				Clear(STRUCT_ALIGNMENT2);
				STRUCT_ALIGNMENT2.aBool := TRUE; STRUCT_ALIGNMENT2.aInt := -1; STRUCT_ALIGNMENT2.aUint := 2;
				STRUCT_ALIGNMENT2.Bools[0] := TRUE; STRUCT_ALIGNMENT2.Bools[3] := TRUE;
				iVarBinSize := ToAryByte(In:=STRUCT_ALIGNMENT2, Order:=_eBYTE_ORDER#_LOW_HIGH, AryOut:=iVarBin[0]);
				Inc(iVarIndex);
			211:
				iVarName := 'STRUCT_ALIGNMENT2_ARR_D1';
				iVarDeclare := 'ARRAY[0..2] OF Alignment2Struct';
				iVarValue := '[{"aBool":true, "aInt":-1, "aUint":2, "Bools":[true,false,false,true]}, {"aBool":false, "aInt":0, "aUint":0, "Bools":[false,false,false,false]}, {"aBool":true, "aInt":-1, "aUint":2, "Bools":[true,false,false,true]}]';
				iVarKsType := 'alignment2_struct_t::alignment2_struct_array_1d(3)';
				iVarKsId := 'struct_alignment2_arr_d1';
				
				Clear(STRUCT_ALIGNMENT2);
				STRUCT_ALIGNMENT2.aBool := TRUE; STRUCT_ALIGNMENT2.aInt := -1; STRUCT_ALIGNMENT2.aUint := 2;
				STRUCT_ALIGNMENT2.Bools[0] := TRUE; STRUCT_ALIGNMENT2.Bools[3] := TRUE;
				Clear(STRUCT_ALIGNMENT2_ARR_D1);
				STRUCT_ALIGNMENT2_ARR_D1[0] := STRUCT_ALIGNMENT2; STRUCT_ALIGNMENT2_ARR_D1[2] := STRUCT_ALIGNMENT2;
				
				iVarBinSize := ToAryByte(In:=STRUCT_ALIGNMENT2_ARR_D1, Order:=_eBYTE_ORDER#_LOW_HIGH, AryOut:=iVarBin[0]);
				iVarIndex := iVarIndex - iVarIndex MOD 10 + 10;

			// Alignment4Struct
			220:
				iVarName := 'STRUCT_ALIGNMENT4';
				iVarDeclare := 'Alignment4Struct';
				iVarValue := '{"aUdint":1, "aDint":-2, "Uints":[3,4], "Bytes":[5,6,7,8]}';
				iVarKsType := 'alignment4_struct_t::alignment4_struct';
				iVarKsId := 'struct_alignment4';
				
				Clear(STRUCT_ALIGNMENT4);
				STRUCT_ALIGNMENT4.aUdint := 1; STRUCT_ALIGNMENT4.aDint := -2;
				STRUCT_ALIGNMENT4.Uints[0] := 3; STRUCT_ALIGNMENT4.Uints[1] := 4;
				STRUCT_ALIGNMENT4.Bytes[0] := 5; STRUCT_ALIGNMENT4.Bytes[1] := 6; STRUCT_ALIGNMENT4.Bytes[2] := 7; STRUCT_ALIGNMENT4.Bytes[3] := 8;
				iVarBinSize := ToAryByte(In:=STRUCT_ALIGNMENT4, Order:=_eBYTE_ORDER#_LOW_HIGH, AryOut:=iVarBin[0]);
				iVarIndex := iVarIndex - iVarIndex MOD 10 + 10;
				
			// Alignment8Struct
			230:
				iVarName := 'STRUCT_ALIGNMENT8';
				iVarDeclare := 'Alignment8Struct';
				iVarValue := '{"aUlint":1, "aLint":-2, "Udints":[3,4], "aAlignment2Struct":{"aBool":true, "aInt":-1, "aUint":2, "Bools":[true,false,false,true]}}';
				iVarKsType := 'alignment8_struct_t::alignment8_struct';
				iVarKsId := 'struct_alignment8';
				
				Clear(STRUCT_ALIGNMENT8);
				STRUCT_ALIGNMENT8.aUlint := 1; STRUCT_ALIGNMENT8.aLint := -2;
				STRUCT_ALIGNMENT8.Udints[0] := 3; STRUCT_ALIGNMENT8.Udints[1] := 4;
				Clear(STRUCT_ALIGNMENT2);
				STRUCT_ALIGNMENT2.aBool := TRUE; STRUCT_ALIGNMENT2.aInt := -1; STRUCT_ALIGNMENT2.aUint := 2;
				STRUCT_ALIGNMENT2.Bools[0] := TRUE; STRUCT_ALIGNMENT2.Bools[3] := TRUE;
				STRUCT_ALIGNMENT8.aAlignment2Struct := STRUCT_ALIGNMENT2;
				iVarBinSize := ToAryByte(In:=STRUCT_ALIGNMENT8, Order:=_eBYTE_ORDER#_LOW_HIGH, AryOut:=iVarBin[0]);
				iVarIndex := iVarIndex - iVarIndex MOD 10 + 10;
			
			// SmallStruct
			240:
				iVarName := 'STRUCT_SMALL_LH';
				iVarDeclare := 'SmallStruct';
				iVarValue := '{"s":"a","u":1}';
				iVarKsType := 'small_struct_t::small_struct';
				iVarKsId := 'struct_small_lh';
				
				Clear(STRUCT_SMALL);
				STRUCT_SMALL.u := 1; STRUCT_SMALL.s := 'a';
				iVarBinSize := ToAryByte(In:=STRUCT_SMALL, Order:=_eBYTE_ORDER#_LOW_HIGH, AryOut:=iVarBin[0]);
				Inc(iVarIndex);
			241:
				iVarName := 'STRUCT_SMALL_ARR_D1_LH';
				iVarDeclare := 'ARRAY[0..2] OF SmallStruct';
				iVarValue := '[{"s":"a","u":1},{"s":"b","u":2},{"s":"c","u":3}]';
				iVarKsType := 'small_struct_t::small_struct_array_1d(3)';
				iVarKsId := 'struct_small_arr_d1_lh';
				
				Clear(STRUCT_SMALL_ARR_D1);
				STRUCT_SMALL_ARR_D1[0].u := 1; STRUCT_SMALL_ARR_D1[0].s := 'a';
				STRUCT_SMALL_ARR_D1[1].u := 2; STRUCT_SMALL_ARR_D1[1].s := 'b';
				STRUCT_SMALL_ARR_D1[2].u := 3; STRUCT_SMALL_ARR_D1[2].s := 'c';
				iVarBinSize := ToAryByte(In:=STRUCT_SMALL_ARR_D1, Order:=_eBYTE_ORDER#_LOW_HIGH, AryOut:=iVarBin[0]);
				Inc(iVarIndex);
			242:
				iVarName := 'STRUCT_SMALL_ARR_D2_LH';
				iVarDeclare := 'ARRAY[0..2,0..2] OF SmallStruct';
				iVarValue := '[[{"s":"a","u":1},{"s":"b","u":2},{"s":"c","u":3}],[{"s":"d","u":4},{"s":"e","u":5},{"s":"f","u":6}],[{"s":"g","u":7},{"s":"h","u":8},{"s":"i","u":9}]]';
				iVarKsType := 'small_struct_t::small_struct_array_2d(3,3)';
				iVarKsId := 'struct_small_arr_d2_lh';
				
				Clear(STRUCT_SMALL_ARR_D2);
				STRUCT_SMALL_ARR_D2[0, 0].u := 1; STRUCT_SMALL_ARR_D2[0, 0].s := 'a';
				STRUCT_SMALL_ARR_D2[0, 1].u := 2; STRUCT_SMALL_ARR_D2[0, 1].s := 'b';
				STRUCT_SMALL_ARR_D2[0, 2].u := 3; STRUCT_SMALL_ARR_D2[0, 2].s := 'c';
				STRUCT_SMALL_ARR_D2[1, 0].u := 4; STRUCT_SMALL_ARR_D2[1, 0].s := 'd';
				STRUCT_SMALL_ARR_D2[1, 1].u := 5; STRUCT_SMALL_ARR_D2[1, 1].s := 'e';
				STRUCT_SMALL_ARR_D2[1, 2].u := 6; STRUCT_SMALL_ARR_D2[1, 2].s := 'f';
				STRUCT_SMALL_ARR_D2[2, 0].u := 7; STRUCT_SMALL_ARR_D2[2, 0].s := 'g';
				STRUCT_SMALL_ARR_D2[2, 1].u := 8; STRUCT_SMALL_ARR_D2[2, 1].s := 'h';
				STRUCT_SMALL_ARR_D2[2, 2].u := 9; STRUCT_SMALL_ARR_D2[2, 2].s := 'i';
				iVarBinSize := ToAryByte(In:=STRUCT_SMALL_ARR_D2, Order:=_eBYTE_ORDER#_LOW_HIGH, AryOut:=iVarBin[0]);
				Inc(iVarIndex);
			243:
				iVarName := 'STRUCT_SMALL_ARR_D3_LH';
				iVarDeclare := 'ARRAY[0..2,0..2,0..2] OF SmallStruct';
				iVarValue := '[[[{"s":"a","u":1},{"s":"b","u":2},{"s":"c","u":3}],[{"s":"d","u":4},{"s":"e","u":5},{"s":"f","u":6}],[{"s":"g","u":7},{"s":"h","u":8},{"s":"i","u":9}]],[[{"s":"j","u":10},{"s":"k","u":11},{"s":"l","u":12}],[{"s":"m","u":13},{"s":"n","u":14},{"s":"o","u":15}],[{"s":"p","u":16},{"s":"q","u":17},{"s":"r","u":18}]],[[{"s":"s","u":19},{"s":"t","u":20},{"s":"u","u":21}],[{"s":"v","u":22},{"s":"w","u":23},{"s":"x","u":24}],[{"s":"y","u":25},{"s":"z","u":26},{"s":"0","u":27}]]]';
				iVarKsType := 'small_struct_t::small_struct_array_3d(3,3,3)';
				iVarKsId := 'struct_small_arr_d3_lh';
				
				Clear(STRUCT_SMALL_ARR_D3);
				STRUCT_SMALL_ARR_D3[0, 0, 0].u := 1; STRUCT_SMALL_ARR_D3[0, 0, 0].s := 'a';
				STRUCT_SMALL_ARR_D3[0, 0, 1].u := 2; STRUCT_SMALL_ARR_D3[0, 0, 1].s := 'b';
				STRUCT_SMALL_ARR_D3[0, 0, 2].u := 3; STRUCT_SMALL_ARR_D3[0, 0, 2].s := 'c';
				STRUCT_SMALL_ARR_D3[0, 1, 0].u := 4; STRUCT_SMALL_ARR_D3[0, 1, 0].s := 'd';
				STRUCT_SMALL_ARR_D3[0, 1, 1].u := 5; STRUCT_SMALL_ARR_D3[0, 1, 1].s := 'e';
				STRUCT_SMALL_ARR_D3[0, 1, 2].u := 6; STRUCT_SMALL_ARR_D3[0, 1, 2].s := 'f';
				STRUCT_SMALL_ARR_D3[0, 2, 0].u := 7; STRUCT_SMALL_ARR_D3[0, 2, 0].s := 'g';
				STRUCT_SMALL_ARR_D3[0, 2, 1].u := 8; STRUCT_SMALL_ARR_D3[0, 2, 1].s := 'h';
				STRUCT_SMALL_ARR_D3[0, 2, 2].u := 9; STRUCT_SMALL_ARR_D3[0, 2, 2].s := 'i';
				STRUCT_SMALL_ARR_D3[1, 0, 0].u := 10; STRUCT_SMALL_ARR_D3[1, 0, 0].s := 'j';
				STRUCT_SMALL_ARR_D3[1, 0, 1].u := 11; STRUCT_SMALL_ARR_D3[1, 0, 1].s := 'k';
				STRUCT_SMALL_ARR_D3[1, 0, 2].u := 12; STRUCT_SMALL_ARR_D3[1, 0, 2].s := 'l';
				STRUCT_SMALL_ARR_D3[1, 1, 0].u := 13; STRUCT_SMALL_ARR_D3[1, 1, 0].s := 'm';
				STRUCT_SMALL_ARR_D3[1, 1, 1].u := 14; STRUCT_SMALL_ARR_D3[1, 1, 1].s := 'n';
				STRUCT_SMALL_ARR_D3[1, 1, 2].u := 15; STRUCT_SMALL_ARR_D3[1, 1, 2].s := 'o';
				STRUCT_SMALL_ARR_D3[1, 2, 0].u := 16; STRUCT_SMALL_ARR_D3[1, 2, 0].s := 'p';
				STRUCT_SMALL_ARR_D3[1, 2, 1].u := 17; STRUCT_SMALL_ARR_D3[1, 2, 1].s := 'q';
				STRUCT_SMALL_ARR_D3[1, 2, 2].u := 18; STRUCT_SMALL_ARR_D3[1, 2, 2].s := 'r';
				STRUCT_SMALL_ARR_D3[2, 0, 0].u := 19; STRUCT_SMALL_ARR_D3[2, 0, 0].s := 's';
				STRUCT_SMALL_ARR_D3[2, 0, 1].u := 20; STRUCT_SMALL_ARR_D3[2, 0, 1].s := 't';
				STRUCT_SMALL_ARR_D3[2, 0, 2].u := 21; STRUCT_SMALL_ARR_D3[2, 0, 2].s := 'u';
				STRUCT_SMALL_ARR_D3[2, 1, 0].u := 22; STRUCT_SMALL_ARR_D3[2, 1, 0].s := 'v';
				STRUCT_SMALL_ARR_D3[2, 1, 1].u := 23; STRUCT_SMALL_ARR_D3[2, 1, 1].s := 'w';
				STRUCT_SMALL_ARR_D3[2, 1, 2].u := 24; STRUCT_SMALL_ARR_D3[2, 1, 2].s := 'x';
				STRUCT_SMALL_ARR_D3[2, 2, 0].u := 25; STRUCT_SMALL_ARR_D3[2, 2, 0].s := 'y';
				STRUCT_SMALL_ARR_D3[2, 2, 1].u := 26; STRUCT_SMALL_ARR_D3[2, 2, 1].s := 'z';
				STRUCT_SMALL_ARR_D3[2, 2, 2].u := 27; STRUCT_SMALL_ARR_D3[2, 2, 2].s := '0';
				iVarBinSize := ToAryByte(In:=STRUCT_SMALL_ARR_D3, Order:=_eBYTE_ORDER#_LOW_HIGH, AryOut:=iVarBin[0]);
				Inc(iVarIndex);
			244:
				iVarName := 'STRUCT_SMALL_ARR_D1_E1_LH';
				iVarDeclare := 'ARRAY[0..0] OF SmallStruct';
				iVarValue := '[{"s":"a","u":1}]';
				iVarKsType := 'small_struct_t::small_struct_array_1d(1)';
				iVarKsId := 'struct_small_arr_d1_e1_lh';
				
				Clear(STRUCT_SMALL_ARR_D1_E1);
				STRUCT_SMALL_ARR_D1_E1[0].u := 1; STRUCT_SMALL_ARR_D1_E1[0].s := 'a';
				iVarBinSize := ToAryByte(In:=STRUCT_SMALL_ARR_D1_E1, Order:=_eBYTE_ORDER#_LOW_HIGH, AryOut:=iVarBin[0]);
				Inc(iVarIndex);
			245:
				iVarName := 'STRUCT_SMALL_ARR_D2_E1_LH';
				iVarDeclare := 'ARRAY[0..0,0..0] OF SmallStruct';
				iVarValue := '[[{"s":"a","u":1}]]';
				iVarKsType := 'small_struct_t::small_struct_array_2d(1,1)';
				iVarKsId := 'struct_small_arr_d2_e1_lh';
				
				Clear(STRUCT_SMALL_ARR_D2_E1);
				STRUCT_SMALL_ARR_D2_E1[0, 0].u := 1; STRUCT_SMALL_ARR_D2_E1[0, 0].s := 'a';
				iVarBinSize := ToAryByte(In:=STRUCT_SMALL_ARR_D2_E1, Order:=_eBYTE_ORDER#_LOW_HIGH, AryOut:=iVarBin[0]);
				Inc(iVarIndex);
			246:
				iVarName := 'STRUCT_SMALL_ARR_D3_E1_LH';
				iVarDeclare := 'ARRAY[0..0,0..0,0..0] OF SmallStruct';
				iVarValue := '[[[{"s":"a","u":1}]]]';
				iVarKsType := 'small_struct_t::small_struct_array_3d(1,1,1)';
				iVarKsId := 'struct_small_arr_d3_e1_lh';
				
				Clear(STRUCT_SMALL_ARR_D3_E1);
				STRUCT_SMALL_ARR_D3_E1[0, 0, 0].u := 1; STRUCT_SMALL_ARR_D3_E1[0, 0, 0].s := 'a';
				iVarBinSize := ToAryByte(In:=STRUCT_SMALL_ARR_D3_E1, Order:=_eBYTE_ORDER#_LOW_HIGH, AryOut:=iVarBin[0]);
				iVarIndex := iVarIndex - iVarIndex MOD 10 + 10;
				
			// PaddedStruct
			250:
				iVarName := 'STRUCT_PADDED_LH';
				iVarDeclare := 'PaddedStruct';
				iVarValue := '{"aUsint":1, "aUint":2, "aSint":-3, "aDint":-4, "aUlint":5, "aBool":true}';
				iVarKsType := 'padded_struct_t::padded_struct';
				iVarKsId := 'struct_padded_lh';
				
				Clear(STRUCT_PADDED);
				STRUCT_PADDED.aUsint := 1; STRUCT_PADDED.aUint := 2; STRUCT_PADDED.aSint := -3;
				STRUCT_PADDED.aDint := -4; STRUCT_PADDED.aUlint := 5; STRUCT_PADDED.aBool := TRUE;
				iVarBinSize := ToAryByte(In:=STRUCT_PADDED, Order:=_eBYTE_ORDER#_LOW_HIGH, AryOut:=iVarBin[0]);
				Inc(iVarIndex);
			251:
				iVarName := 'STRUCT_PADDED_ARR_D1_LH';
				iVarDeclare := 'ARRAY[0..2] OF PaddedStruct';
				iVarValue := '[{"aUsint":1, "aUint":2, "aSint":-3, "aDint":-4, "aUlint":5, "aBool":true}, {"aUsint":6, "aUint":7, "aSint":-8, "aDint":-9, "aUlint":10, "aBool":false}, {"aUsint":11, "aUint":12, "aSint":-13, "aDint":-14, "aUlint":15, "aBool":true}]';
				iVarKsType := 'padded_struct_t::padded_struct_array_1d(3)';
				iVarKsId := 'struct_padded_arr_d1_lh';
				
				Clear(STRUCT_PADDED_ARR_D1);
				STRUCT_PADDED_ARR_D1[0].aUsint := 1; STRUCT_PADDED_ARR_D1[0].aUint := 2; STRUCT_PADDED_ARR_D1[0].aSint := -3;
				STRUCT_PADDED_ARR_D1[0].aDint := -4; STRUCT_PADDED_ARR_D1[0].aUlint := 5; STRUCT_PADDED_ARR_D1[0].aBool := TRUE;
				STRUCT_PADDED_ARR_D1[1].aUsint := 6; STRUCT_PADDED_ARR_D1[1].aUint := 7; STRUCT_PADDED_ARR_D1[1].aSint := -8;
				STRUCT_PADDED_ARR_D1[1].aDint := -9; STRUCT_PADDED_ARR_D1[1].aUlint := 10; STRUCT_PADDED_ARR_D1[1].aBool := FALSE;
				STRUCT_PADDED_ARR_D1[2].aUsint := 11; STRUCT_PADDED_ARR_D1[2].aUint := 12; STRUCT_PADDED_ARR_D1[2].aSint := -13;
				STRUCT_PADDED_ARR_D1[2].aDint := -14; STRUCT_PADDED_ARR_D1[2].aUlint := 15; STRUCT_PADDED_ARR_D1[2].aBool := TRUE;
				iVarBinSize := ToAryByte(In:=STRUCT_PADDED_ARR_D1, Order:=_eBYTE_ORDER#_LOW_HIGH, AryOut:=iVarBin[0]);
				Inc(iVarIndex);
			252:
				iVarName := 'STRUCT_PADDED_ARR_D1_E1_LH';
				iVarDeclare := 'ARRAY[0..0] OF PaddedStruct';
				iVarValue := '[{"aUsint":1, "aUint":2, "aSint":-3, "aDint":-4, "aUlint":5, "aBool":true}]';
				iVarKsType := 'padded_struct_t::padded_struct_array_1d(1)';
				iVarKsId := 'struct_padded_arr_d1_e1_lh';
				
				Clear(STRUCT_PADDED_ARR_D1_E1);
				STRUCT_PADDED_ARR_D1_E1[0].aUsint := 1; STRUCT_PADDED_ARR_D1_E1[0].aUint := 2; STRUCT_PADDED_ARR_D1_E1[0].aSint := -3;
				STRUCT_PADDED_ARR_D1_E1[0].aDint := -4; STRUCT_PADDED_ARR_D1_E1[0].aUlint := 5; STRUCT_PADDED_ARR_D1_E1[0].aBool := TRUE;
				iVarBinSize := ToAryByte(In:=STRUCT_PADDED_ARR_D1_E1, Order:=_eBYTE_ORDER#_LOW_HIGH, AryOut:=iVarBin[0]);
				Inc(iVarIndex);
			253:
				iVarName := 'STRUCT_PADDED_ARR_D2_E1_LH';
				iVarDeclare := 'ARRAY[0..0,0..0] OF PaddedStruct';
				iVarValue := '[[{"aUsint":1, "aUint":2, "aSint":-3, "aDint":-4, "aUlint":5, "aBool":true}]]';
				iVarKsType := 'padded_struct_t::padded_struct_array_2d(1,1)';
				iVarKsId := 'struct_padded_arr_d2_e1_lh';
				
				Clear(STRUCT_PADDED_ARR_D2_E1);
				STRUCT_PADDED_ARR_D2_E1[0, 0].aUsint := 1; STRUCT_PADDED_ARR_D2_E1[0, 0].aUint := 2; STRUCT_PADDED_ARR_D2_E1[0, 0].aSint := -3;
				STRUCT_PADDED_ARR_D2_E1[0, 0].aDint := -4; STRUCT_PADDED_ARR_D2_E1[0, 0].aUlint := 5; STRUCT_PADDED_ARR_D2_E1[0, 0].aBool := TRUE;
				iVarBinSize := ToAryByte(In:=STRUCT_PADDED_ARR_D2_E1, Order:=_eBYTE_ORDER#_LOW_HIGH, AryOut:=iVarBin[0]);
				Inc(iVarIndex);
			254:
				iVarName := 'STRUCT_PADDED_ARR_D3_E1_LH';
				iVarDeclare := 'ARRAY[0..0,0..0,0..0] OF PaddedStruct';
				iVarValue := '[[[{"aUsint":1, "aUint":2, "aSint":-3, "aDint":-4, "aUlint":5, "aBool":true}]]]';
				iVarKsType := 'padded_struct_t::padded_struct_array_3d(1,1,1)';
				iVarKsId := 'struct_padded_arr_d3_e1_lh';
				
				Clear(STRUCT_PADDED_ARR_D3_E1);
				STRUCT_PADDED_ARR_D3_E1[0, 0, 0].aUsint := 1; STRUCT_PADDED_ARR_D3_E1[0, 0, 0].aUint := 2; STRUCT_PADDED_ARR_D3_E1[0, 0, 0].aSint := -3;
				STRUCT_PADDED_ARR_D3_E1[0, 0, 0].aDint := -4; STRUCT_PADDED_ARR_D3_E1[0, 0, 0].aUlint := 5; STRUCT_PADDED_ARR_D3_E1[0, 0, 0].aBool := TRUE;
				iVarBinSize := ToAryByte(In:=STRUCT_PADDED_ARR_D3_E1, Order:=_eBYTE_ORDER#_LOW_HIGH, AryOut:=iVarBin[0]);
				iVarIndex := iVarIndex - iVarIndex MOD 10 + 10;

			// UnionStruct
			260:
				iVarName := 'STRUCT_UNION_LH';
				iVarDeclare := 'UnionStruct';
				// Since Union is not supported, the values ​​of each field are listed separately.
				iVarValue := '{"Alignment1Unions":[{"Bytes":[1,2,3,4]},{"Bytes":[5,6,7,8]}], "Alignment2Unions":[{"aBool":true,"Words":[9,10]}, {"aBool":true,"Words":[11,12]}], "aAlignment4Union":{"Bytes":[13,0,0,0],"Dwords":[13,14]}, "aAlignment8Union":{"Words":[15,0,0,0],"aLword":15}}';
				iVarKsType := 'union_struct_t::union_struct';
				iVarKsId := 'union_struct_lh';
				
				Clear(STRUCT_UNION);
				STRUCT_UNION.Alignment1Unions[0].Bytes[0] := 1; STRUCT_UNION.Alignment1Unions[0].Bytes[1] := 2; STRUCT_UNION.Alignment1Unions[0].Bytes[2] := 3; STRUCT_UNION.Alignment1Unions[0].Bytes[3] := 4;
				STRUCT_UNION.Alignment1Unions[1].Bytes[0] := 5; STRUCT_UNION.Alignment1Unions[1].Bytes[1] := 6; STRUCT_UNION.Alignment1Unions[1].Bytes[2] := 7; STRUCT_UNION.Alignment1Unions[1].Bytes[3] := 8;
				STRUCT_UNION.Alignment2Unions[0].Words[0] := 9; STRUCT_UNION.Alignment2Unions[0].Words[1] := 10;
				STRUCT_UNION.Alignment2Unions[1].Words[0] := 11; STRUCT_UNION.Alignment2Unions[1].Words[1] := 12;
				STRUCT_UNION.aAlignment4Union.Dwords[0] := 13; STRUCT_UNION.aAlignment4Union.Dwords[1] := 14;
				STRUCT_UNION.aAlignment8Union.aLword := 15;
				
				iVarBinSize := ToAryByte(In:=STRUCT_UNION, Order:=_eBYTE_ORDER#_LOW_HIGH, AryOut:=iVarBin[0]);
				Inc(iVarIndex);
			261:
				iVarName := 'STRUCT_UNION_ARR_D1_LH';
				iVarDeclare := 'ARRAY[0..2] OF UnionStruct';
				// Since Union is not supported, the values ​​of each field are listed separately.
				iVarValue := '[{"Alignment1Unions":[{"Bytes":[1,2,3,4]},{"Bytes":[5,6,7,8]}], "Alignment2Unions":[{"aBool":true,"Words":[9,10]}, {"aBool":true,"Words":[11,12]}], "aAlignment4Union":{"Bytes":[13,0,0,0],"Dwords":[13,14]}, "aAlignment8Union":{"Words":[15,0,0,0],"aLword":15}},{"Alignment1Unions":[{"Bytes":[16,17,18,19]},{"Bytes":[20,21,22,23]}], "Alignment2Unions":[{"aBool":false,"Words":[24,25]}, {"aBool":false,"Words":[26,27]}], "aAlignment4Union":{"Bytes":[28,0,0,0],"Dwords":[28,29]}, "aAlignment8Union":{"Words":[30,0,0,0],"aLword":30}},{"Alignment1Unions":[{"Bytes":[31,32,33,34]},{"Bytes":[35,36,37,38]}], "Alignment2Unions":[{"aBool":true,"Words":[39,40]}, {"aBool":true,"Words":[41,42]}], "aAlignment4Union":{"Bytes":[43,0,0,0],"Dwords":[43,44]}, "aAlignment8Union":{"Words":[45,0,0,0],"aLword":45}}]';
				iVarKsType := 'union_struct_t::union_struct_array_1d(3)';
				iVarKsId := 'union_struct_arr_d1_lh';
				
				Clear(STRUCT_UNION);
				STRUCT_UNION_ARR_D1[0].Alignment1Unions[0].Bytes[0] := 1; STRUCT_UNION_ARR_D1[0].Alignment1Unions[0].Bytes[1] := 2; STRUCT_UNION_ARR_D1[0].Alignment1Unions[0].Bytes[2] := 3; STRUCT_UNION_ARR_D1[0].Alignment1Unions[0].Bytes[3] := 4;
				STRUCT_UNION_ARR_D1[0].Alignment1Unions[1].Bytes[0] := 5; STRUCT_UNION_ARR_D1[0].Alignment1Unions[1].Bytes[1] := 6; STRUCT_UNION_ARR_D1[0].Alignment1Unions[1].Bytes[2] := 7; STRUCT_UNION_ARR_D1[0].Alignment1Unions[1].Bytes[3] := 8;
				STRUCT_UNION_ARR_D1[0].Alignment2Unions[0].Words[0] := 9; STRUCT_UNION_ARR_D1[0].Alignment2Unions[0].Words[1] := 10;
				STRUCT_UNION_ARR_D1[0].Alignment2Unions[1].Words[0] := 11; STRUCT_UNION_ARR_D1[0].Alignment2Unions[1].Words[1] := 12;
				STRUCT_UNION_ARR_D1[0].aAlignment4Union.Dwords[0] := 13; STRUCT_UNION_ARR_D1[0].aAlignment4Union.Dwords[1] := 14;
				STRUCT_UNION_ARR_D1[0].aAlignment8Union.aLword := 15;

				STRUCT_UNION_ARR_D1[1].Alignment1Unions[0].Bytes[0] := 16; STRUCT_UNION_ARR_D1[1].Alignment1Unions[0].Bytes[1] := 17; STRUCT_UNION_ARR_D1[1].Alignment1Unions[0].Bytes[2] := 18; STRUCT_UNION_ARR_D1[1].Alignment1Unions[0].Bytes[3] := 19;
				STRUCT_UNION_ARR_D1[1].Alignment1Unions[1].Bytes[0] := 20; STRUCT_UNION_ARR_D1[1].Alignment1Unions[1].Bytes[1] := 21; STRUCT_UNION_ARR_D1[1].Alignment1Unions[1].Bytes[2] := 22; STRUCT_UNION_ARR_D1[1].Alignment1Unions[1].Bytes[3] := 23;
				STRUCT_UNION_ARR_D1[1].Alignment2Unions[0].Words[0] := 24; STRUCT_UNION_ARR_D1[1].Alignment2Unions[0].Words[1] := 25;
				STRUCT_UNION_ARR_D1[1].Alignment2Unions[1].Words[0] := 26; STRUCT_UNION_ARR_D1[1].Alignment2Unions[1].Words[1] := 27;
				STRUCT_UNION_ARR_D1[1].aAlignment4Union.Dwords[0] := 28; STRUCT_UNION_ARR_D1[1].aAlignment4Union.Dwords[1] := 29;
				STRUCT_UNION_ARR_D1[1].aAlignment8Union.aLword := 30;

				STRUCT_UNION_ARR_D1[2].Alignment1Unions[0].Bytes[0] := 31; STRUCT_UNION_ARR_D1[2].Alignment1Unions[0].Bytes[1] := 32; STRUCT_UNION_ARR_D1[2].Alignment1Unions[0].Bytes[2] := 33; STRUCT_UNION_ARR_D1[2].Alignment1Unions[0].Bytes[3] := 34;
				STRUCT_UNION_ARR_D1[2].Alignment1Unions[1].Bytes[0] := 35; STRUCT_UNION_ARR_D1[2].Alignment1Unions[1].Bytes[1] := 36; STRUCT_UNION_ARR_D1[2].Alignment1Unions[1].Bytes[2] := 37; STRUCT_UNION_ARR_D1[2].Alignment1Unions[1].Bytes[3] := 38;
				STRUCT_UNION_ARR_D1[2].Alignment2Unions[0].Words[0] := 39; STRUCT_UNION_ARR_D1[2].Alignment2Unions[0].Words[1] := 40;
				STRUCT_UNION_ARR_D1[2].Alignment2Unions[1].Words[0] := 41; STRUCT_UNION_ARR_D1[2].Alignment2Unions[1].Words[1] := 42;
				STRUCT_UNION_ARR_D1[2].aAlignment4Union.Dwords[0] := 43; STRUCT_UNION_ARR_D1[2].aAlignment4Union.Dwords[1] := 44;
				STRUCT_UNION_ARR_D1[2].aAlignment8Union.aLword := 45;

				iVarBinSize := ToAryByte(In:=STRUCT_UNION_ARR_D1, Order:=_eBYTE_ORDER#_LOW_HIGH, AryOut:=iVarBin[0]);
				Inc(iVarIndex);
			262:
				iVarName := 'STRUCT_UNION_ARR_D1_E1_LH';
				iVarDeclare := 'ARRAY[0..0] OF UnionStruct';
				// Since Union is not supported, the values ​​of each field are listed separately.
				iVarValue := '[{"Alignment1Unions":[{"Bytes":[1,2,3,4]},{"Bytes":[5,6,7,8]}], "Alignment2Unions":[{"aBool":true,"Words":[9,10]}, {"aBool":true,"Words":[11,12]}], "aAlignment4Union":{"Bytes":[13,0,0,0],"Dwords":[13,14]}, "aAlignment8Union":{"Words":[15,0,0,0],"aLword":15}}]';
				iVarKsType := 'union_struct_t::union_struct_array_1d(1)';
				iVarKsId := 'union_struct_arr_d1_e1_lh';
				
				Clear(STRUCT_UNION_ARR_D1_E1);
				STRUCT_UNION_ARR_D1_E1[0].Alignment1Unions[0].Bytes[0] := 1; STRUCT_UNION_ARR_D1_E1[0].Alignment1Unions[0].Bytes[1] := 2; STRUCT_UNION_ARR_D1_E1[0].Alignment1Unions[0].Bytes[2] := 3; STRUCT_UNION_ARR_D1_E1[0].Alignment1Unions[0].Bytes[3] := 4;
				STRUCT_UNION_ARR_D1_E1[0].Alignment1Unions[1].Bytes[0] := 5; STRUCT_UNION_ARR_D1_E1[0].Alignment1Unions[1].Bytes[1] := 6; STRUCT_UNION_ARR_D1_E1[0].Alignment1Unions[1].Bytes[2] := 7; STRUCT_UNION_ARR_D1_E1[0].Alignment1Unions[1].Bytes[3] := 8;
				STRUCT_UNION_ARR_D1_E1[0].Alignment2Unions[0].Words[0] := 9; STRUCT_UNION_ARR_D1_E1[0].Alignment2Unions[0].Words[1] := 10;
				STRUCT_UNION_ARR_D1_E1[0].Alignment2Unions[1].Words[0] := 11; STRUCT_UNION_ARR_D1_E1[0].Alignment2Unions[1].Words[1] := 12;
				STRUCT_UNION_ARR_D1_E1[0].aAlignment4Union.Dwords[0] := 13; STRUCT_UNION_ARR_D1_E1[0].aAlignment4Union.Dwords[1] := 14;
				STRUCT_UNION_ARR_D1_E1[0].aAlignment8Union.aLword := 15;

				iVarBinSize := ToAryByte(In:=STRUCT_UNION_ARR_D1_E1, Order:=_eBYTE_ORDER#_LOW_HIGH, AryOut:=iVarBin[0]);
				Inc(iVarIndex);
			263:
				iVarName := 'STRUCT_UNION_ARR_D2_E1_LH';
				iVarDeclare := 'ARRAY[0..0,0..0] OF UnionStruct';
				// Since Union is not supported, the values ​​of each field are listed separately.
				iVarValue := '[[{"Alignment1Unions":[{"Bytes":[1,2,3,4]},{"Bytes":[5,6,7,8]}], "Alignment2Unions":[{"aBool":true,"Words":[9,10]}, {"aBool":true,"Words":[11,12]}], "aAlignment4Union":{"Bytes":[13,0,0,0],"Dwords":[13,14]}, "aAlignment8Union":{"Words":[15,0,0,0],"aLword":15}}]]';
				iVarKsType := 'union_struct_t::union_struct_array_2d(1,1)';
				iVarKsId := 'union_struct_arr_d2_e1_lh';
				
				Clear(STRUCT_UNION_ARR_D2_E1);
				STRUCT_UNION_ARR_D2_E1[0, 0].Alignment1Unions[0].Bytes[0] := 1; STRUCT_UNION_ARR_D2_E1[0, 0].Alignment1Unions[0].Bytes[1] := 2; STRUCT_UNION_ARR_D2_E1[0, 0].Alignment1Unions[0].Bytes[2] := 3; STRUCT_UNION_ARR_D2_E1[0, 0].Alignment1Unions[0].Bytes[3] := 4;
				STRUCT_UNION_ARR_D2_E1[0, 0].Alignment1Unions[1].Bytes[0] := 5; STRUCT_UNION_ARR_D2_E1[0, 0].Alignment1Unions[1].Bytes[1] := 6; STRUCT_UNION_ARR_D2_E1[0, 0].Alignment1Unions[1].Bytes[2] := 7; STRUCT_UNION_ARR_D2_E1[0, 0].Alignment1Unions[1].Bytes[3] := 8;
				STRUCT_UNION_ARR_D2_E1[0, 0].Alignment2Unions[0].Words[0] := 9; STRUCT_UNION_ARR_D2_E1[0, 0].Alignment2Unions[0].Words[1] := 10;
				STRUCT_UNION_ARR_D2_E1[0, 0].Alignment2Unions[1].Words[0] := 11; STRUCT_UNION_ARR_D2_E1[0, 0].Alignment2Unions[1].Words[1] := 12;
				STRUCT_UNION_ARR_D2_E1[0, 0].aAlignment4Union.Dwords[0] := 13; STRUCT_UNION_ARR_D2_E1[0, 0].aAlignment4Union.Dwords[1] := 14;
				STRUCT_UNION_ARR_D2_E1[0, 0].aAlignment8Union.aLword := 15;
				iVarBinSize := ToAryByte(In:=STRUCT_UNION_ARR_D2_E1, Order:=_eBYTE_ORDER#_LOW_HIGH, AryOut:=iVarBin[0]);
				Inc(iVarIndex);
			264:
				iVarName := 'STRUCT_UNION_ARR_D3_E1_LH';
				iVarDeclare := 'ARRAY[0..0,0..0,0..0] OF UnionStruct';
				// Since Union is not supported, the values ​​of each field are listed separately.
				iVarValue := '[[[{"Alignment1Unions":[{"Bytes":[1,2,3,4]},{"Bytes":[5,6,7,8]}], "Alignment2Unions":[{"aBool":true,"Words":[9,10]}, {"aBool":true,"Words":[11,12]}], "aAlignment4Union":{"Bytes":[13,0,0,0],"Dwords":[13,14]}, "aAlignment8Union":{"Words":[15,0,0,0],"aLword":15}}]]]';
				iVarKsType := 'union_struct_t::union_struct_array_3d(1,1,1)';
				iVarKsId := 'union_struct_arr_d3_e1_lh';
				
				Clear(STRUCT_UNION_ARR_D3_E1);
				STRUCT_UNION_ARR_D3_E1[0, 0, 0].Alignment1Unions[0].Bytes[0] := 1; STRUCT_UNION_ARR_D3_E1[0, 0, 0].Alignment1Unions[0].Bytes[1] := 2; STRUCT_UNION_ARR_D3_E1[0, 0, 0].Alignment1Unions[0].Bytes[2] := 3; STRUCT_UNION_ARR_D3_E1[0, 0, 0].Alignment1Unions[0].Bytes[3] := 4;
				STRUCT_UNION_ARR_D3_E1[0, 0, 0].Alignment1Unions[1].Bytes[0] := 5; STRUCT_UNION_ARR_D3_E1[0, 0, 0].Alignment1Unions[1].Bytes[1] := 6; STRUCT_UNION_ARR_D3_E1[0, 0, 0].Alignment1Unions[1].Bytes[2] := 7; STRUCT_UNION_ARR_D3_E1[0, 0, 0].Alignment1Unions[1].Bytes[3] := 8;
				STRUCT_UNION_ARR_D3_E1[0, 0, 0].Alignment2Unions[0].Words[0] := 9; STRUCT_UNION_ARR_D3_E1[0, 0, 0].Alignment2Unions[0].Words[1] := 10;
				STRUCT_UNION_ARR_D3_E1[0, 0, 0].Alignment2Unions[1].Words[0] := 11; STRUCT_UNION_ARR_D3_E1[0, 0, 0].Alignment2Unions[1].Words[1] := 12;
				STRUCT_UNION_ARR_D3_E1[0, 0, 0].aAlignment4Union.Dwords[0] := 13; STRUCT_UNION_ARR_D3_E1[0, 0, 0].aAlignment4Union.Dwords[1] := 14;
				STRUCT_UNION_ARR_D3_E1[0, 0, 0].aAlignment8Union.aLword := 15;
				iVarBinSize := ToAryByte(In:=STRUCT_UNION_ARR_D3_E1, Order:=_eBYTE_ORDER#_LOW_HIGH, AryOut:=iVarBin[0]);
				Inc(iVarIndex);
				iVarIndex := 300;

			// Union
			// Alignment1Union
			300:
				iVarName := 'UNION_ALIGNMENT1_LH';
				iVarDeclare := 'Alignment1Union';
				iVarValue := '{"Bytes":[0,1,2,3]}';
				iVarKsType := 'alignment1_union_t::alignment1_union';
				iVarKsId := 'union_alignment1_lh';
				
				Clear(UNION_ALIGNMENT1.Bytes);
				UNION_ALIGNMENT1.Bytes[0] := 0; UNION_ALIGNMENT1.Bytes[1] := 1; UNION_ALIGNMENT1.Bytes[2] := 2; UNION_ALIGNMENT1.Bytes[3] := 3;
				iVarBinSize := ToAryByte(In:=UNION_ALIGNMENT1.Bytes, Order:=_eBYTE_ORDER#_LOW_HIGH, AryOut:=iVarBin[0]);
				Inc(iVarIndex);
			301:
				iVarName := 'UNION_ALIGNMENT1_ARR_D1_LH';
				iVarDeclare := 'ARRAY[0..2] OF Alignment1Union';
				iVarValue := '[{"Bytes":[0,1,2,3]},{"Bytes":[5,6,7,8]},{"Bytes":[9,10,11,12]}]';
				iVarKsType := 'alignment1_union_t::alignment1_union_array_1d(3)';
				iVarKsId := 'union_alignment1_arr_d1_lh';
				
				Clear(UNION_ALIGNMENT1_ARR_D1);
				UNION_ALIGNMENT1_ARR_D1.Unions[0].Bytes[0] := 0; UNION_ALIGNMENT1_ARR_D1.Unions[0].Bytes[1] := 1; UNION_ALIGNMENT1_ARR_D1.Unions[0].Bytes[2] := 2; UNION_ALIGNMENT1_ARR_D1.Unions[0].Bytes[3] := 3;
				UNION_ALIGNMENT1_ARR_D1.Unions[1].Bytes[0] := 5; UNION_ALIGNMENT1_ARR_D1.Unions[1].Bytes[1] := 6; UNION_ALIGNMENT1_ARR_D1.Unions[1].Bytes[2] := 7; UNION_ALIGNMENT1_ARR_D1.Unions[1].Bytes[3] := 8;
				UNION_ALIGNMENT1_ARR_D1.Unions[2].Bytes[0] := 9; UNION_ALIGNMENT1_ARR_D1.Unions[2].Bytes[1] := 10; UNION_ALIGNMENT1_ARR_D1.Unions[2].Bytes[2] := 11; UNION_ALIGNMENT1_ARR_D1.Unions[2].Bytes[3] := 12;
				iVarBinSize := ToAryByte(In:=UNION_ALIGNMENT1_ARR_D1, Order:=_eBYTE_ORDER#_LOW_HIGH, AryOut:=iVarBin[0]);
				iVarIndex := iVarIndex - iVarIndex MOD 10 + 10;

			// Alignment2Union
			310:
				iVarName := 'UNION_ALIGNMENT2_LH';
				iVarDeclare := 'Alignment2Union';
				iVarValue := '{"aBool":true,"Words":[1,0]}';
				iVarKsType := 'alignment2_union_t::alignment2_union';
				iVarKsId := 'union_alignment2_lh';
				
				Clear(UNION_ALIGNMENT2.Words);
				UNION_ALIGNMENT2.aBool := TRUE;
				iVarBinSize := ToAryByte(In:=UNION_ALIGNMENT2.Words, Order:=_eBYTE_ORDER#_LOW_HIGH, AryOut:=iVarBin[0]);
				Inc(iVarIndex);
			311:
				iVarName := 'UNION_ALIGNMENT2_ARR_D1_LH';
				iVarDeclare := 'ARRAY[0..2] OF Alignment2Union';
				iVarValue := '[{"aBool":true,"Words":[1,0]}, {"aBool":false,"Words":[2,0]}, {"aBool":true,"Words":[3,8]}]';
				iVarKsType := 'alignment2_union_t::alignment2_union_array_1d(3)';
				iVarKsId := 'union_alignment2_arr_d1_lh';
				
				// Define it as a struct and pack it to enable conversion.
				Clear(UNION_ALIGNMENT2_ARR_D1);
				UNION_ALIGNMENT2_ARR_D1.Unions[0].aBool := TRUE;
				UNION_ALIGNMENT2_ARR_D1.Unions[1].Words[0] := 2;
				UNION_ALIGNMENT2_ARR_D1.Unions[2].Words[0] := 3; UNION_ALIGNMENT2_ARR_D1.Unions[2].Words[1] := 8;
				iVarBinSize := ToAryByte(In:=UNION_ALIGNMENT2_ARR_D1, Order:=_eBYTE_ORDER#_LOW_HIGH, AryOut:=iVarBin[0]);
				Inc(iVarIndex);
			312:
				iVarName := 'UNION_ALIGNMENT2_ARR_D2_LH';
				iVarDeclare := 'ARRAY[0..2,0..2] OF Alignment2Union';
				iVarValue := '[[{"aBool":true,"Words":[1,0]}, {"aBool":false,"Words":[2,0]}, {"aBool":true,"Words":[3,8]}],[{"aBool":false,"Words":[4,0]}, {"aBool":true,"Words":[5,0]}, {"aBool":false,"Words":[6,16]}],[{"aBool":true,"Words":[7,0]}, {"aBool":false,"Words":[8,0]}, {"aBool":true,"Words":[9,32]}]]';
				iVarKsType := 'alignment2_union_t::alignment2_union_array_2d(3,3)';
				iVarKsId := 'union_alignment2_arr_d2_lh';
				
				// Define it as a struct and pack it to enable conversion.
				Clear(UNION_ALIGNMENT2_ARR_D2);
				UNION_ALIGNMENT2_ARR_D2.Unions[0, 0].aBool := TRUE;
				UNION_ALIGNMENT2_ARR_D2.Unions[0, 1].Words[0] := 2;
				UNION_ALIGNMENT2_ARR_D2.Unions[0, 2].Words[0] := 3; UNION_ALIGNMENT2_ARR_D2.Unions[0, 2].Words[1] := 8;
				UNION_ALIGNMENT2_ARR_D2.Unions[1, 0].Words[0] := 4; UNION_ALIGNMENT2_ARR_D2.Unions[1, 0].Words[1] := 0;
				UNION_ALIGNMENT2_ARR_D2.Unions[1, 1].Words[0] := 5; UNION_ALIGNMENT2_ARR_D2.Unions[1, 1].Words[1] := 0;
				UNION_ALIGNMENT2_ARR_D2.Unions[1, 2].Words[0] := 6; UNION_ALIGNMENT2_ARR_D2.Unions[1, 2].Words[1] := 16;
				UNION_ALIGNMENT2_ARR_D2.Unions[2, 0].Words[0] := 7; UNION_ALIGNMENT2_ARR_D2.Unions[2, 0].Words[1] := 0;
				UNION_ALIGNMENT2_ARR_D2.Unions[2, 1].Words[0] := 8; UNION_ALIGNMENT2_ARR_D2.Unions[2, 1].Words[1] := 0;
				UNION_ALIGNMENT2_ARR_D2.Unions[2, 2].Words[0] := 9; UNION_ALIGNMENT2_ARR_D2.Unions[2, 2].Words[1] := 32;
				iVarBinSize := ToAryByte(In:=UNION_ALIGNMENT2_ARR_D2, Order:=_eBYTE_ORDER#_LOW_HIGH, AryOut:=iVarBin[0]);
				Inc(iVarIndex);
			313:
				iVarName := 'UNION_ALIGNMENT2_ARR_D3_LH';
				iVarDeclare := 'ARRAY[0..2,0..2,0..2] OF Alignment2Union';
				iVarValue := '[[[{"aBool":true,"Words":[1,0]}, {"aBool":false,"Words":[2,0]}, {"aBool":true,"Words":[3,8]}],[{"aBool":false,"Words":[4,0]}, {"aBool":true,"Words":[5,0]}, {"aBool":false,"Words":[6,16]}],[{"aBool":true,"Words":[7,0]}, {"aBool":false,"Words":[8,0]}, {"aBool":true,"Words":[9,32]}]],[[{"aBool":false,"Words":[0,0]}, {"aBool":false,"Words":[10,0]}, {"aBool":true,"Words":[11,64]}],[{"aBool":false,"Words":[12,0]}, {"aBool":true,"Words":[13,0]}, {"aBool":false,"Words":[14,128]}],[{"aBool":true,"Words":[15,0]}, {"aBool":false,"Words":[16,0]}, {"aBool":true,"Words":[17,256]}]],[[{"aBool":true,"Words":[1,0]}, {"aBool":false,"Words":[18,0]}, {"aBool":true,"Words":[19,512]}],[{"aBool":false,"Words":[20,0]}, {"aBool":true,"Words":[21,0]}, {"aBool":false,"Words":[22,1024]}],[{"aBool":true,"Words":[23,0]}, {"aBool":false,"Words":[24,0]}, {"aBool":true,"Words":[25,2048]}]]';
				iVarKsType := 'alignment2_union_t::alignment2_union_array_3d(3,3,3)';
				iVarKsId := 'union_alignment2_arr_d3_lh';
				
				// Define it as a struct and pack it to enable conversion.
				Clear(UNION_ALIGNMENT2_ARR_D3);
				UNION_ALIGNMENT2_ARR_D3.Unions[0, 0, 0].aBool := TRUE;
				UNION_ALIGNMENT2_ARR_D3.Unions[0, 0, 1].Words[0] := 2; UNION_ALIGNMENT2_ARR_D3.Unions[0, 0, 1].Words[1] := 0;
				UNION_ALIGNMENT2_ARR_D3.Unions[0, 0, 2].Words[0] := 3; UNION_ALIGNMENT2_ARR_D3.Unions[0, 0, 2].Words[1] := 8;
				UNION_ALIGNMENT2_ARR_D3.Unions[0, 1, 0].Words[0] := 4; UNION_ALIGNMENT2_ARR_D3.Unions[0, 1, 0].Words[1] := 0;
				UNION_ALIGNMENT2_ARR_D3.Unions[0, 1, 1].Words[0] := 5; UNION_ALIGNMENT2_ARR_D3.Unions[0, 1, 1].Words[1] := 0;
				UNION_ALIGNMENT2_ARR_D3.Unions[0, 1, 2].Words[0] := 6; UNION_ALIGNMENT2_ARR_D3.Unions[0, 1, 2].Words[1] := 16;
				UNION_ALIGNMENT2_ARR_D3.Unions[0, 2, 0].Words[0] := 7; UNION_ALIGNMENT2_ARR_D3.Unions[0, 2, 0].Words[1] := 0;
				UNION_ALIGNMENT2_ARR_D3.Unions[0, 2, 1].Words[0] := 8; UNION_ALIGNMENT2_ARR_D3.Unions[0, 2, 1].Words[1] := 0;
				UNION_ALIGNMENT2_ARR_D3.Unions[0, 2, 2].Words[0] := 9; UNION_ALIGNMENT2_ARR_D3.Unions[0, 2, 2].Words[1] := 32;

				UNION_ALIGNMENT2_ARR_D3.Unions[1, 0, 0].aBool := FALSE;
				UNION_ALIGNMENT2_ARR_D3.Unions[1, 0, 1].Words[0] := 10; UNION_ALIGNMENT2_ARR_D3.Unions[1, 0, 1].Words[1] := 0;
				UNION_ALIGNMENT2_ARR_D3.Unions[1, 0, 2].Words[0] := 11; UNION_ALIGNMENT2_ARR_D3.Unions[1, 0, 2].Words[1] := 64;
				UNION_ALIGNMENT2_ARR_D3.Unions[1, 1, 0].Words[0] := 12; UNION_ALIGNMENT2_ARR_D3.Unions[1, 1, 0].Words[1] := 0;
				UNION_ALIGNMENT2_ARR_D3.Unions[1, 1, 1].Words[0] := 13; UNION_ALIGNMENT2_ARR_D3.Unions[1, 1, 1].Words[1] := 0;
				UNION_ALIGNMENT2_ARR_D3.Unions[1, 1, 2].Words[0] := 14; UNION_ALIGNMENT2_ARR_D3.Unions[1, 1, 2].Words[1] := 128;
				UNION_ALIGNMENT2_ARR_D3.Unions[1, 2, 0].Words[0] := 15; UNION_ALIGNMENT2_ARR_D3.Unions[1, 2, 0].Words[1] := 0;
				UNION_ALIGNMENT2_ARR_D3.Unions[1, 2, 1].Words[0] := 16; UNION_ALIGNMENT2_ARR_D3.Unions[1, 2, 1].Words[1] := 0;
				UNION_ALIGNMENT2_ARR_D3.Unions[1, 2, 2].Words[0] := 17; UNION_ALIGNMENT2_ARR_D3.Unions[1, 2, 2].Words[1] := 256;

				UNION_ALIGNMENT2_ARR_D3.Unions[2, 0, 0].aBool := TRUE;
				UNION_ALIGNMENT2_ARR_D3.Unions[2, 0, 1].Words[0] := 18; UNION_ALIGNMENT2_ARR_D3.Unions[2, 0, 1].Words[1] := 0;
				UNION_ALIGNMENT2_ARR_D3.Unions[2, 0, 2].Words[0] := 19; UNION_ALIGNMENT2_ARR_D3.Unions[2, 0, 2].Words[1] := 512;
				UNION_ALIGNMENT2_ARR_D3.Unions[2, 1, 0].Words[0] := 20; UNION_ALIGNMENT2_ARR_D3.Unions[2, 1, 0].Words[1] := 0;
				UNION_ALIGNMENT2_ARR_D3.Unions[2, 1, 1].Words[0] := 21; UNION_ALIGNMENT2_ARR_D3.Unions[2, 1, 1].Words[1] := 0;
				UNION_ALIGNMENT2_ARR_D3.Unions[2, 1, 2].Words[0] := 22; UNION_ALIGNMENT2_ARR_D3.Unions[2, 1, 2].Words[1] := 1024;
				UNION_ALIGNMENT2_ARR_D3.Unions[2, 2, 0].Words[0] := 23; UNION_ALIGNMENT2_ARR_D3.Unions[2, 2, 0].Words[1] := 0;
				UNION_ALIGNMENT2_ARR_D3.Unions[2, 2, 1].Words[0] := 24; UNION_ALIGNMENT2_ARR_D3.Unions[2, 2, 1].Words[1] := 0;
				UNION_ALIGNMENT2_ARR_D3.Unions[2, 2, 2].Words[0] := 25; UNION_ALIGNMENT2_ARR_D3.Unions[2, 2, 2].Words[1] := 2048;

				iVarBinSize := ToAryByte(In:=UNION_ALIGNMENT2_ARR_D3, Order:=_eBYTE_ORDER#_LOW_HIGH, AryOut:=iVarBin[0]);
				Inc(iVarIndex);
			314:
				iVarName := 'UNION_ALIGNMENT2_ARR_D1_E1_LH';
				iVarDeclare := 'ARRAY[0..0] OF Alignment2Union';
				iVarValue := '[{"aBool":true,"Words":[1,0]}]';
				iVarKsType := 'alignment2_union_t::alignment2_union_array_1d(1)';
				iVarKsId := 'union_alignment2_arr_d1_e1_lh';
				
				// Define it as a struct and pack it to enable conversion.
				Clear(UNION_ALIGNMENT2_ARR_D1_E1);
				UNION_ALIGNMENT2_ARR_D1_E1.Unions[0].aBool := TRUE;
				iVarBinSize := ToAryByte(In:=UNION_ALIGNMENT2_ARR_D1_E1, Order:=_eBYTE_ORDER#_LOW_HIGH, AryOut:=iVarBin[0]);
				Inc(iVarIndex);
			315:
				iVarName := 'UNION_ALIGNMENT2_ARR_D2_E1_LH';
				iVarDeclare := 'ARRAY[0..0,0..0] OF Alignment2Union';
				iVarValue := '[[{"aBool":true,"Words":[1,0]}]]';
				iVarKsType := 'alignment2_union_t::alignment2_union_array_2d(1,1)';
				iVarKsId := 'union_alignment2_arr_d2_e1_lh';
				
				// Define it as a struct and pack it to enable conversion.
				Clear(UNION_ALIGNMENT2_ARR_D2_E1);
				UNION_ALIGNMENT2_ARR_D2_E1.Unions[0, 0].aBool := TRUE;
				iVarBinSize := ToAryByte(In:=UNION_ALIGNMENT2_ARR_D2_E1, Order:=_eBYTE_ORDER#_LOW_HIGH, AryOut:=iVarBin[0]);
				Inc(iVarIndex);
			316:
				iVarName := 'UNION_ALIGNMENT2_ARR_D3_E1_LH';
				iVarDeclare := 'ARRAY[0..0,0..0,0..0] OF Alignment2Union';
				iVarValue := '[[[{"aBool":true,"Words":[1,0]}]]]';
				iVarKsType := 'alignment2_union_t::alignment2_union_array_3d(1,1,1)';
				iVarKsId := 'union_alignment2_arr_d3_e1_lh';
				
				// Define it as a struct and pack it to enable conversion.
				Clear(UNION_ALIGNMENT2_ARR_D3_E1);
				UNION_ALIGNMENT2_ARR_D3_E1.Unions[0, 0, 0].aBool := TRUE;
				iVarBinSize := ToAryByte(In:=UNION_ALIGNMENT2_ARR_D3_E1, Order:=_eBYTE_ORDER#_LOW_HIGH, AryOut:=iVarBin[0]);
				iVarIndex := iVarIndex - iVarIndex MOD 10 + 10;

			// Alignment4Union
			320:
				iVarName := 'UNION_ALIGNMENT4_LH';
				iVarDeclare := 'Alignment4Union';
				iVarValue := '{"Bytes":[1,0,0,0],"Dwords":[1,2]}';
				iVarKsType := 'alignment4_union_t::alignment4_union';
				iVarKsId := 'union_alignment4_lh';
				
				Clear(UNION_ALIGNMENT4.Dwords);
				UNION_ALIGNMENT4.Dwords[0] := 1; UNION_ALIGNMENT4.Dwords[1] := 2;
				iVarBinSize := ToAryByte(In:=UNION_ALIGNMENT4.Dwords, Order:=_eBYTE_ORDER#_LOW_HIGH, AryOut:=iVarBin[0]);
				Inc(iVarIndex);
			321:
				iVarName := 'UNION_ALIGNMENT4_ARR_D1_E1_LH';
				iVarDeclare := 'Alignment4Union';
				iVarValue := '[{"Bytes":[1,0,0,0],"Dwords":[1,2]}]';
				iVarKsType := 'alignment4_union_t::alignment4_union_array_1d(1)';
				iVarKsId := 'union_alignment4_arr_d1_e1_lh';
				
				// Define it as a struct and pack it to enable conversion.
				Clear(UNION_ALIGNMENT4_ARR_D1_E1);
				UNION_ALIGNMENT4_ARR_D1_E1.Unions[0].Dwords[0] := 1; UNION_ALIGNMENT4_ARR_D1_E1.Unions[0].Dwords[1] := 2;
				iVarBinSize := ToAryByte(In:=UNION_ALIGNMENT4_ARR_D1_E1, Order:=_eBYTE_ORDER#_LOW_HIGH, AryOut:=iVarBin[0]);
				Inc(iVarIndex);
			322:
				iVarName := 'UNION_ALIGNMENT4_ARR_D2_E1_LH';
				iVarDeclare := 'Alignment4Union';
				iVarValue := '[[{"Bytes":[1,0,0,0],"Dwords":[1,2]}]]';
				iVarKsType := 'alignment4_union_t::alignment4_union_array_2d(1,1)';
				iVarKsId := 'union_alignment4_arr_d2_e1_lh';
				
				// Define it as a struct and pack it to enable conversion.
				Clear(UNION_ALIGNMENT4_ARR_D2_E1);
				UNION_ALIGNMENT4_ARR_D2_E1.Unions[0, 0].Dwords[0] := 1; UNION_ALIGNMENT4_ARR_D2_E1.Unions[0, 0].Dwords[1] := 2;
				iVarBinSize := ToAryByte(In:=UNION_ALIGNMENT4_ARR_D2_E1, Order:=_eBYTE_ORDER#_LOW_HIGH, AryOut:=iVarBin[0]);
				Inc(iVarIndex);
			323:
				iVarName := 'UNION_ALIGNMENT4_ARR_D3_E1_LH';
				iVarDeclare := 'Alignment4Union';
				iVarValue := '[[[{"Bytes":[1,0,0,0],"Dwords":[1,2]}]]]';
				iVarKsType := 'alignment4_union_t::alignment4_union_array_3d(1,1,1)';
				iVarKsId := 'union_alignment4_arr_d3_e1_lh';
				
				// Define it as a struct and pack it to enable conversion.
				Clear(UNION_ALIGNMENT4_ARR_D3_E1);
				UNION_ALIGNMENT4_ARR_D3_E1.Unions[0, 0, 0].Dwords[0] := 1; UNION_ALIGNMENT4_ARR_D3_E1.Unions[0, 0, 0].Dwords[1] := 2;
				iVarBinSize := ToAryByte(In:=UNION_ALIGNMENT4_ARR_D3_E1, Order:=_eBYTE_ORDER#_LOW_HIGH, AryOut:=iVarBin[0]);
				iVarIndex := iVarIndex - iVarIndex MOD 10 + 10;

			// Alignment8Union
			330:
				iVarName := 'UNION_ALIGNMENT8_LH';
				iVarDeclare := 'Alignment8Union';
				iVarValue := '{"Words":[1,0,0,0],"aLword":1}';
				iVarKsType := 'alignment8_union_t::alignment8_union';
				iVarKsId := 'union_alignment8_lh';
				
				Clear(UNION_ALIGNMENT8.aLword);
				UNION_ALIGNMENT8.aLword := 1;
				iVarBinSize := ToAryByte(In:=UNION_ALIGNMENT8.aLword, Order:=_eBYTE_ORDER#_LOW_HIGH, AryOut:=iVarBin[0]);
				Inc(iVarIndex);
			331:
				iVarName := 'UNION_ALIGNMENT8_ARR_D1_E1_LH';
				iVarDeclare := 'Alignment8Union';
				iVarValue := '[{"Words":[1,0,0,0],"aLword":1}]';
				iVarKsType := 'alignment8_union_t::alignment8_union_array_1d(1)';
				iVarKsId := 'union_alignment8_arr_d1_e1_lh';
				
				// Define it as a struct and pack it to enable conversion.
				Clear(UNION_ALIGNMENT8_ARR_D1_E1);
				UNION_ALIGNMENT8_ARR_D1_E1.Unions[0].aLword := 1;
				iVarBinSize := ToAryByte(In:=UNION_ALIGNMENT8_ARR_D1_E1, Order:=_eBYTE_ORDER#_LOW_HIGH, AryOut:=iVarBin[0]);
				Inc(iVarIndex);
			332:
				iVarName := 'UNION_ALIGNMENT8_ARR_D2_E1_LH';
				iVarDeclare := 'Alignment8Union';
				iVarValue := '[[{"Words":[1,0,0,0],"aLword":1}]]';
				iVarKsType := 'alignment8_union_t::alignment8_union_array_2d(1,1)';
				iVarKsId := 'union_alignment8_arr_d2_e1_lh';
				
				// Define it as a struct and pack it to enable conversion.
				Clear(UNION_ALIGNMENT8_ARR_D2_E1);
				UNION_ALIGNMENT8_ARR_D2_E1.Unions[0, 0].aLword := 1;
				iVarBinSize := ToAryByte(In:=UNION_ALIGNMENT8_ARR_D2_E1, Order:=_eBYTE_ORDER#_LOW_HIGH, AryOut:=iVarBin[0]);
				Inc(iVarIndex);
			333:
				iVarName := 'UNION_ALIGNMENT8_ARR_D3_E1_LH';
				iVarDeclare := 'Alignment8Union';
				iVarValue := '[[[{"Words":[1,0,0,0],"aLword":1}]]]';
				iVarKsType := 'alignment8_union_t::alignment8_union_array_3d(1,1,1)';
				iVarKsId := 'union_alignment8_arr_d3_e1_lh';
				
				// Define it as a struct and pack it to enable conversion.
				Clear(UNION_ALIGNMENT8_ARR_D3_E1);
				UNION_ALIGNMENT8_ARR_D3_E1.Unions[0, 0, 0].aLword := 1;
				iVarBinSize := ToAryByte(In:=UNION_ALIGNMENT8_ARR_D3_E1, Order:=_eBYTE_ORDER#_LOW_HIGH, AryOut:=iVarBin[0]);
				iVarIndex := iVarIndex - iVarIndex MOD 10 + 10;

			// ComplexStruct
			340:
				iVarName := 'STRUCT_COMPLEX_LH';
				iVarDeclare := 'ComplexStruct';
				iVarValue := '{"aUsint":128,"Alignment2Structs":[{"aBool":true,"aInt":1,"aUint":2,"Bools":[true,false,true,false]},{"aBool":false,"aInt":3,"aUint":4,"Bools":[false,true,false,true]}],"aAlignment4Union":{"Bytes":[5,0,0,0],"Dwords":[5,6]},"aBool":true,"Lints":[-7,8],"aEnum":1}';
				iVarKsType := 'complex_struct_t::complex_struct';
				iVarKsId := 'struct_complex_lh';
				
				Clear(STRUCT_COMPLEX);
				STRUCT_COMPLEX.aUsint := 128;
				Clear(STRUCT_ALIGNMENT2);
				STRUCT_ALIGNMENT2.aBool := TRUE; STRUCT_ALIGNMENT2.aInt := 1; STRUCT_ALIGNMENT2.aUint := 2; STRUCT_ALIGNMENT2.Bools[0] := TRUE; STRUCT_ALIGNMENT2.Bools[2] := TRUE;
				STRUCT_COMPLEX.Alignment2Structs[0] := STRUCT_ALIGNMENT2;
				Clear(STRUCT_ALIGNMENT2);
				STRUCT_ALIGNMENT2.aBool := FALSE; STRUCT_ALIGNMENT2.aInt := 3; STRUCT_ALIGNMENT2.aUint := 4; STRUCT_ALIGNMENT2.Bools[1] := TRUE; STRUCT_ALIGNMENT2.Bools[3] := TRUE;
				STRUCT_COMPLEX.Alignment2Structs[1] := STRUCT_ALIGNMENT2;
				Clear(UNION_ALIGNMENT4.Dwords);
				UNION_ALIGNMENT4.Dwords[0] := 5; UNION_ALIGNMENT4.Dwords[1] := 6;
				STRUCT_COMPLEX.aAlignment4Union.Dwords := UNION_ALIGNMENT4.Dwords;
				STRUCT_COMPLEX.aBool := TRUE;
				STRUCT_COMPLEX.Lints[0] := -7; STRUCT_COMPLEX.Lints[1] := 8;
				STRUCT_COMPLEX.aEnum := TestEnum#TE_E1;
				
				iVarBinSize := ToAryByte(In:=STRUCT_COMPLEX, Order:=_eBYTE_ORDER#_LOW_HIGH, AryOut:=iVarBin[0]);
				iVarIndex := iVarIndex + 10;

			// Nest3Struct
			350:
				iVarName := 'STRUCT_NEST3_LH';
				iVarDeclare := 'Nest3Struct';
				iVarValue := '{"aSmallStruct":{"u":5,"s":"L3"},"aNest2Struct":{"aSmallStruct":{"u":3,"s":"L2"},"aNest1Struct":{"aSmallStruct":{"u":1,"s":"L1"},"aInt":-2},"aDint":-4},"aLint":-6}';
				iVarKsType := 'nest3_struct_t::nest3_struct';
				iVarKsId := 'struct_nest3_lh';
				
				Clear(STRUCT_SMALL);
				STRUCT_SMALL.u := 1;
				STRUCT_SMALL.s := 'L1';
				Clear(STRUCT_NEST1);
				STRUCT_NEST1.aSmallStruct := STRUCT_SMALL;
				STRUCT_NEST1.aInt := -2;
				Clear(STRUCT_NEST2);
				STRUCT_NEST2.aNest1Struct := STRUCT_NEST1;
				Clear(STRUCT_SMALL);
				STRUCT_SMALL.u := 3;
				STRUCT_SMALL.s := 'L2';
				STRUCT_NEST2.aSmallStruct := STRUCT_SMALL;
				STRUCT_NEST2.aDint := -4;
				Clear(STRUCT_NEST3);
				STRUCT_NEST3.aNest2Struct := STRUCT_NEST2;
				Clear(STRUCT_SMALL);
				STRUCT_SMALL.u := 5;
				STRUCT_SMALL.s := 'L3';
				STRUCT_NEST3.aSmallStruct := STRUCT_SMALL;
				STRUCT_NEST3.aLint := -6;
								
				iVarBinSize := ToAryByte(In:=STRUCT_NEST3, Order:=_eBYTE_ORDER#_LOW_HIGH, AryOut:=iVarBin[0]);
				iVarIndex := iVarIndex + 10;

			// ExampleStruct
			360:
				iVarName := 'STRUCT_EXAMPLE_LH';
				iVarDeclare := 'ExampleStruct';
				iVarValue := '{"Acc":3.513, "Trq":17.255, "Vel":6.965, "StatusCode":3840}';
				iVarKsType := 'example_struct';
				iVarKsId := 'example_struct_lh';
				
				Clear(STRUCT_EXAMPLE);
				STRUCT_EXAMPLE.Acc := 3.513;
				STRUCT_EXAMPLE.Trq := 17.255;
				STRUCT_EXAMPLE.Vel := 6.965;
				STRUCT_EXAMPLE.StatusCode := DWORD#16#0F00;
								
				iVarBinSize := ToAryByte(In:=STRUCT_EXAMPLE, Order:=_eBYTE_ORDER#_LOW_HIGH, AryOut:=iVarBin[0]);
				iVarIndex := iVarIndex + 10;

			// ExampleUnion
			370:
				iVarName := 'STRUCT_UNION_LH';
				iVarDeclare := 'ExampleUnion';
				iVarValue := '{"StatusFlags":[false,false,false,false,true,false,false,false,  false,false,false,false,false,true,false,false],"SegmentedStatusCodes":[8208,32832],"StatusCode":2151686160}';
				iVarKsType := 'example_union';
				iVarKsId := 'example_union_lh';
				
				Clear(UNION_EXAMPLE.StatusCode);
				UNION_EXAMPLE.StatusCode := DWORD#2#10000000_01000000_00100000_00010000;
								
				iVarBinSize := ToAryByte(In:=UNION_EXAMPLE.StatusCode, Order:=_eBYTE_ORDER#_LOW_HIGH, AryOut:=iVarBin[0]);
				iVarIndex := iVarIndex + 10;
		ELSE
				iVarIndex := 1000;			
		END_CASE;
		
		IF iVarIndex < 1000 THEN		
			Inc(iState);
		ELSE
			iState := iState + 7;
		END_IF;
	23: // Writes var list as an array.
		IF iCurrentVarIndex < 1 THEN
			RingBuffer_writeStr(Context:=iBufferContext,
								Buffer:=iBuffer,
								In:='@($n');
		END_IF;
		
		RingBuffer_writeStr(Context:=iBufferContext,
							Buffer:=iBuffer,
							In:=CONCAT('# size: ', UINT_TO_STRING(iVarBinSize), ' declare: ', iVarDeclare, '$n'));
		RingBuffer_writeStr(Context:=iBufferContext,
							Buffer:=iBuffer,
							In:=CONCAT(
									CONCAT('@{Key = $'', iVarName, '$''),
									CONCAT('; Json = $'', iVarValue, '$'; Declare = $'', iVarDeclare, '$''),
									CONCAT('; KsType = $'', iVarKsType, '$''),
									CONCAT('; KsId = $'', iVarKsId, '$''),
									'; Hex = '
									));
		RingBuffer_writeAsHexStr(Context:=iBufferContext,
								 Buffer:=iBuffer,
								 In:=iVarBin,
								 Head:=0,
								 Size:=iVarBinSize,
								 Prefix:='0x',
								 Join:=', ');
		RingBuffer_writeStr(Context:=iBufferContext,
							Buffer:=iBuffer,
							In:='};$n');

		IF iCurrentVarIndex >= 370 THEN
			RingBuffer_writeStr(Context:=iBufferContext,
								Buffer:=iBuffer,
								In:=');');
		END_IF;
		
		Inc(iState);
	24:
		IF NOT \\stfreakjp\fileio\FileStreamWriter_isFlushing(iFileWriterContext) THEN
			Inc(iState);
		END_IF;
	25: // Writes each var files.
		iFileWriteVar(Execute:=FALSE, WriteVar:=iVarBin);
		
		iVarFilePath := CONCAT(WRITE_VAR_BASE_PATH, iVarName, '.bin');
		iFileWriteVar.FileName := iVarFilePath;
		iFileWriteVar.OverWrite := TRUE;
		
		Inc(iState);
	26:
		CASE iCurrentVarIndex OF
			// USINT
			0: iFileWriteVar(Execute:=TRUE, WriteVar:=USINT_ARR_D1);
			1: iFileWriteVar(Execute:=TRUE, WriteVar:=USINT_ARR_D2);
			2: iFileWriteVar(Execute:=TRUE, WriteVar:=USINT_ARR_D3);
			3: iFileWriteVar(Execute:=TRUE, WriteVar:=USINT_ARR_D1_E1);
			4: iFileWriteVar(Execute:=TRUE, WriteVar:=USINT_ARR_D2_E1);
			5: iFileWriteVar(Execute:=TRUE, WriteVar:=USINT_ARR_D3_E1);

			// UINT
			10: iFileWriteVar(Execute:=TRUE, WriteVar:=UINT_ARR_D1);
			11: iFileWriteVar(Execute:=TRUE, WriteVar:=UINT_ARR_D2);
			12: iFileWriteVar(Execute:=TRUE, WriteVar:=UINT_ARR_D3);
			13: iFileWriteVar(Execute:=TRUE, WriteVar:=UINT_ARR_D1_E1);
			14: iFileWriteVar(Execute:=TRUE, WriteVar:=UINT_ARR_D2_E1);
			15: iFileWriteVar(Execute:=TRUE, WriteVar:=UINT_ARR_D3_E1);

			// UDINT
			20: iFileWriteVar(Execute:=TRUE, WriteVar:=UDINT_ARR_D1);
			21: iFileWriteVar(Execute:=TRUE, WriteVar:=UDINT_ARR_D2);
			22: iFileWriteVar(Execute:=TRUE, WriteVar:=UDINT_ARR_D3);
			23: iFileWriteVar(Execute:=TRUE, WriteVar:=UDINT_ARR_D1_E1);
			24: iFileWriteVar(Execute:=TRUE, WriteVar:=UDINT_ARR_D2_E1);
			25: iFileWriteVar(Execute:=TRUE, WriteVar:=UDINT_ARR_D3_E1);

			// ULINT
			30: iFileWriteVar(Execute:=TRUE, WriteVar:=ULINT_ARR_D1);
			31: iFileWriteVar(Execute:=TRUE, WriteVar:=ULINT_ARR_D2);
			32: iFileWriteVar(Execute:=TRUE, WriteVar:=ULINT_ARR_D3);
			33: iFileWriteVar(Execute:=TRUE, WriteVar:=ULINT_ARR_D1_E1);
			34: iFileWriteVar(Execute:=TRUE, WriteVar:=ULINT_ARR_D2_E1);
			35: iFileWriteVar(Execute:=TRUE, WriteVar:=ULINT_ARR_D3_E1);

			// SINT
			40: iFileWriteVar(Execute:=TRUE, WriteVar:=SINT_ARR_D1);
			41: iFileWriteVar(Execute:=TRUE, WriteVar:=SINT_ARR_D2);
			42: iFileWriteVar(Execute:=TRUE, WriteVar:=SINT_ARR_D3);
			43: iFileWriteVar(Execute:=TRUE, WriteVar:=SINT_ARR_D1_E1);
			44: iFileWriteVar(Execute:=TRUE, WriteVar:=SINT_ARR_D2_E1);
			45: iFileWriteVar(Execute:=TRUE, WriteVar:=SINT_ARR_D3_E1);

			// INT
			50: iFileWriteVar(Execute:=TRUE, WriteVar:=INT_ARR_D1);
			51: iFileWriteVar(Execute:=TRUE, WriteVar:=INT_ARR_D2);
			52: iFileWriteVar(Execute:=TRUE, WriteVar:=INT_ARR_D3);
			53: iFileWriteVar(Execute:=TRUE, WriteVar:=INT_ARR_D1_E1);
			54: iFileWriteVar(Execute:=TRUE, WriteVar:=INT_ARR_D2_E1);
			55: iFileWriteVar(Execute:=TRUE, WriteVar:=INT_ARR_D3_E1);

			// DINT
			60: iFileWriteVar(Execute:=TRUE, WriteVar:=DINT_ARR_D1);
			61: iFileWriteVar(Execute:=TRUE, WriteVar:=DINT_ARR_D2);
			62: iFileWriteVar(Execute:=TRUE, WriteVar:=DINT_ARR_D3);
			63: iFileWriteVar(Execute:=TRUE, WriteVar:=DINT_ARR_D1_E1);
			64: iFileWriteVar(Execute:=TRUE, WriteVar:=DINT_ARR_D2_E1);
			65: iFileWriteVar(Execute:=TRUE, WriteVar:=DINT_ARR_D3_E1);

			// LINT
			70: iFileWriteVar(Execute:=TRUE, WriteVar:=LINT_ARR_D1);
			71: iFileWriteVar(Execute:=TRUE, WriteVar:=LINT_ARR_D2);
			72: iFileWriteVar(Execute:=TRUE, WriteVar:=LINT_ARR_D3);
			73: iFileWriteVar(Execute:=TRUE, WriteVar:=LINT_ARR_D1_E1);
			74: iFileWriteVar(Execute:=TRUE, WriteVar:=LINT_ARR_D2_E1);
			75: iFileWriteVar(Execute:=TRUE, WriteVar:=LINT_ARR_D3_E1);

			// BYTE
			80: iFileWriteVar(Execute:=TRUE, WriteVar:=BYTE_ARR_D1);
			81: iFileWriteVar(Execute:=TRUE, WriteVar:=BYTE_ARR_D2);
			82: iFileWriteVar(Execute:=TRUE, WriteVar:=BYTE_ARR_D3);
			83: iFileWriteVar(Execute:=TRUE, WriteVar:=BYTE_ARR_D1_E1);
			84: iFileWriteVar(Execute:=TRUE, WriteVar:=BYTE_ARR_D2_E1);
			85: iFileWriteVar(Execute:=TRUE, WriteVar:=BYTE_ARR_D3_E1);

			// WORD
			90: iFileWriteVar(Execute:=TRUE, WriteVar:=WORD_ARR_D1);
			91: iFileWriteVar(Execute:=TRUE, WriteVar:=WORD_ARR_D2);
			92: iFileWriteVar(Execute:=TRUE, WriteVar:=WORD_ARR_D3);
			93: iFileWriteVar(Execute:=TRUE, WriteVar:=WORD_ARR_D1_E1);
			94: iFileWriteVar(Execute:=TRUE, WriteVar:=WORD_ARR_D2_E1);
			95: iFileWriteVar(Execute:=TRUE, WriteVar:=WORD_ARR_D3_E1);

			// DWORD
			100: iFileWriteVar(Execute:=TRUE, WriteVar:=DWORD_ARR_D1);
			101: iFileWriteVar(Execute:=TRUE, WriteVar:=DWORD_ARR_D2);
			102: iFileWriteVar(Execute:=TRUE, WriteVar:=DWORD_ARR_D3);
			103: iFileWriteVar(Execute:=TRUE, WriteVar:=DWORD_ARR_D1_E1);
			104: iFileWriteVar(Execute:=TRUE, WriteVar:=DWORD_ARR_D2_E1);
			105: iFileWriteVar(Execute:=TRUE, WriteVar:=DWORD_ARR_D3_E1);

			// LWORD
			110: iFileWriteVar(Execute:=TRUE, WriteVar:=LWORD_ARR_D1);
			111: iFileWriteVar(Execute:=TRUE, WriteVar:=LWORD_ARR_D2);
			112: iFileWriteVar(Execute:=TRUE, WriteVar:=LWORD_ARR_D3);
			113: iFileWriteVar(Execute:=TRUE, WriteVar:=LWORD_ARR_D1_E1);
			114: iFileWriteVar(Execute:=TRUE, WriteVar:=LWORD_ARR_D2_E1);
			115: iFileWriteVar(Execute:=TRUE, WriteVar:=LWORD_ARR_D3_E1);

			// REAL
			120: iFileWriteVar(Execute:=TRUE, WriteVar:=REAL_ARR_D1);
			121: iFileWriteVar(Execute:=TRUE, WriteVar:=REAL_ARR_D2);
			122: iFileWriteVar(Execute:=TRUE, WriteVar:=REAL_ARR_D3);
			123: iFileWriteVar(Execute:=TRUE, WriteVar:=REAL_ARR_D1_E1);
			124: iFileWriteVar(Execute:=TRUE, WriteVar:=REAL_ARR_D2_E1);
			125: iFileWriteVar(Execute:=TRUE, WriteVar:=REAL_ARR_D3_E1);

			// LREAL
			130: iFileWriteVar(Execute:=TRUE, WriteVar:=LREAL_ARR_D1);
			131: iFileWriteVar(Execute:=TRUE, WriteVar:=LREAL_ARR_D2);
			132: iFileWriteVar(Execute:=TRUE, WriteVar:=LREAL_ARR_D3);
			133: iFileWriteVar(Execute:=TRUE, WriteVar:=LREAL_ARR_D1_E1);
			134: iFileWriteVar(Execute:=TRUE, WriteVar:=LREAL_ARR_D2_E1);
			135: iFileWriteVar(Execute:=TRUE, WriteVar:=LREAL_ARR_D3_E1);

			// STRING
			140: iFileWriteVar(Execute:=TRUE, WriteVar:=STRING_N2);
			141: iFileWriteVar(Execute:=TRUE, WriteVar:=STRING_N2);
			142: iFileWriteVar(Execute:=TRUE, WriteVar:=STRING_N16);
			143: iFileWriteVar(Execute:=TRUE, WriteVar:=STRING_N16);
			144: iFileWriteVar(Execute:=TRUE, WriteVar:=STRING_N16);
			145: iFileWriteVar(Execute:=TRUE, WriteVar:=STRING_N16);
			146: iFileWriteVar(Execute:=TRUE, WriteVar:=STRING_N16);
			147: iFileWriteVar(Execute:=TRUE, WriteVar:=STRING_N16);
			148: iFileWriteVar(Execute:=TRUE, WriteVar:=STRING_N16);
			149: iFileWriteVar(Execute:=TRUE, WriteVar:=STRING_N16);

			// BOOL
			150: iFileWriteVar(Execute:=TRUE, WriteVar:=BOOL_ARR_D1);
			151: iFileWriteVar(Execute:=TRUE, WriteVar:=BOOL_ARR_D2);
			152: iFileWriteVar(Execute:=TRUE, WriteVar:=BOOL_ARR_D3);
			153: iFileWriteVar(Execute:=TRUE, WriteVar:=BOOL_ARR_D1_E1);
			154: iFileWriteVar(Execute:=TRUE, WriteVar:=BOOL_ARR_D2_E1);
			155: iFileWriteVar(Execute:=TRUE, WriteVar:=BOOL_ARR_D3_E1);

			// TIME
			160: iFileWriteVar(Execute:=TRUE, WriteVar:=TIME_ARR_D1);
			161: iFileWriteVar(Execute:=TRUE, WriteVar:=TIME_ARR_D2);
			162: iFileWriteVar(Execute:=TRUE, WriteVar:=TIME_ARR_D3);
			163: iFileWriteVar(Execute:=TRUE, WriteVar:=TIME_ARR_D1_E1);
			164: iFileWriteVar(Execute:=TRUE, WriteVar:=TIME_ARR_D2_E1);
			165: iFileWriteVar(Execute:=TRUE, WriteVar:=TIME_ARR_D3_E1);

			// DATE
			170: iFileWriteVar(Execute:=TRUE, WriteVar:=DATE_ARR_D1);
			171: iFileWriteVar(Execute:=TRUE, WriteVar:=DATE_ARR_D2);
			172: iFileWriteVar(Execute:=TRUE, WriteVar:=DATE_ARR_D3);
			173: iFileWriteVar(Execute:=TRUE, WriteVar:=DATE_ARR_D1_E1);
			174: iFileWriteVar(Execute:=TRUE, WriteVar:=DATE_ARR_D2_E1);
			175: iFileWriteVar(Execute:=TRUE, WriteVar:=DATE_ARR_D3_E1);

			// TIME_OF_DAY
			180: iFileWriteVar(Execute:=TRUE, WriteVar:=TOD_ARR_D1);
			181: iFileWriteVar(Execute:=TRUE, WriteVar:=TOD_ARR_D2);
			182: iFileWriteVar(Execute:=TRUE, WriteVar:=TOD_ARR_D3);
			183: iFileWriteVar(Execute:=TRUE, WriteVar:=TOD_ARR_D1_E1);
			184: iFileWriteVar(Execute:=TRUE, WriteVar:=TOD_ARR_D2_E1);
			185: iFileWriteVar(Execute:=TRUE, WriteVar:=TOD_ARR_D3_E1);

			// DATE_AND_TIME
			190: iFileWriteVar(Execute:=TRUE, WriteVar:=DT_ARR_D1);
			191: iFileWriteVar(Execute:=TRUE, WriteVar:=DT_ARR_D2);
			192: iFileWriteVar(Execute:=TRUE, WriteVar:=DT_ARR_D3);
			193: iFileWriteVar(Execute:=TRUE, WriteVar:=DT_ARR_D1_E1);
			194: iFileWriteVar(Execute:=TRUE, WriteVar:=DT_ARR_D2_E1);
			195: iFileWriteVar(Execute:=TRUE, WriteVar:=DT_ARR_D3_E1);

			// STRUCT
			// Alignment1Struct
			200: iFileWriteVar(Execute:=TRUE, WriteVar:=STRUCT_ALIGNMENT1);
			201: iFileWriteVar(Execute:=TRUE, WriteVar:=STRUCT_ALIGNMENT1_ARR_D1);
			202: iFileWriteVar(Execute:=TRUE, WriteVar:=STRUCT_ALIGNMENT1_ARR_D1_E1);
			203: iFileWriteVar(Execute:=TRUE, WriteVar:=STRUCT_ALIGNMENT1_ARR_D2_E1);
			204: iFileWriteVar(Execute:=TRUE, WriteVar:=STRUCT_ALIGNMENT1_ARR_D3_E1);

			// Alignment2Struct
			210: iFileWriteVar(Execute:=TRUE, WriteVar:=STRUCT_ALIGNMENT2);
			211: iFileWriteVar(Execute:=TRUE, WriteVar:=STRUCT_ALIGNMENT2_ARR_D1);
			212: iFileWriteVar(Execute:=TRUE, WriteVar:=STRUCT_ALIGNMENT2_ARR_D1_E1);
			213: iFileWriteVar(Execute:=TRUE, WriteVar:=STRUCT_ALIGNMENT2_ARR_D2_E1);
			214: iFileWriteVar(Execute:=TRUE, WriteVar:=STRUCT_ALIGNMENT2_ARR_D3_E1);

			// Alignment4Struct
			220: iFileWriteVar(Execute:=TRUE, WriteVar:=STRUCT_ALIGNMENT4);
(*			221: iFileWriteVar(Execute:=TRUE, WriteVar:=STRUCT_ALIGNMENT4_ARR_D1);
			222: iFileWriteVar(Execute:=TRUE, WriteVar:=STRUCT_ALIGNMENT4_ARR_D1_E1);
			223: iFileWriteVar(Execute:=TRUE, WriteVar:=STRUCT_ALIGNMENT4_ARR_D2_E1);
			224: iFileWriteVar(Execute:=TRUE, WriteVar:=STRUCT_ALIGNMENT4_ARR_D3_E1);*)

			// Alignment8Struct
			230: iFileWriteVar(Execute:=TRUE, WriteVar:=STRUCT_ALIGNMENT8);
(*			231: iFileWriteVar(Execute:=TRUE, WriteVar:=STRUCT_ALIGNMENT8_ARR_D1);
			232: iFileWriteVar(Execute:=TRUE, WriteVar:=STRUCT_ALIGNMENT8_ARR_D1_E1);
			233: iFileWriteVar(Execute:=TRUE, WriteVar:=STRUCT_ALIGNMENT8_ARR_D2_E1);
			234: iFileWriteVar(Execute:=TRUE, WriteVar:=STRUCT_ALIGNMENT8_ARR_D3_E1);*)

			// SmallStruct
			240: iFileWriteVar(Execute:=TRUE, WriteVar:=STRUCT_SMALL);
			241: iFileWriteVar(Execute:=TRUE, WriteVar:=STRUCT_SMALL_ARR_D1);
			242: iFileWriteVar(Execute:=TRUE, WriteVar:=STRUCT_SMALL_ARR_D2);
			243: iFileWriteVar(Execute:=TRUE, WriteVar:=STRUCT_SMALL_ARR_D3);
			244: iFileWriteVar(Execute:=TRUE, WriteVar:=STRUCT_SMALL_ARR_D1_E1);
			245: iFileWriteVar(Execute:=TRUE, WriteVar:=STRUCT_SMALL_ARR_D2_E1);
			246: iFileWriteVar(Execute:=TRUE, WriteVar:=STRUCT_SMALL_ARR_D3_E1);

			// PaddedStruct
			250: iFileWriteVar(Execute:=TRUE, WriteVar:=STRUCT_PADDED);
			251: iFileWriteVar(Execute:=TRUE, WriteVar:=STRUCT_PADDED_ARR_D1);
			252: iFileWriteVar(Execute:=TRUE, WriteVar:=STRUCT_PADDED_ARR_D1_E1);
			253: iFileWriteVar(Execute:=TRUE, WriteVar:=STRUCT_PADDED_ARR_D2_E1);
			254: iFileWriteVar(Execute:=TRUE, WriteVar:=STRUCT_PADDED_ARR_D3_E1);

			// UnionStruct
			260: iFileWriteVar(Execute:=TRUE, WriteVar:=STRUCT_UNION);
			261: iFileWriteVar(Execute:=TRUE, WriteVar:=STRUCT_UNION_ARR_D1);
			262: iFileWriteVar(Execute:=TRUE, WriteVar:=STRUCT_UNION_ARR_D1_E1);
			263: iFileWriteVar(Execute:=TRUE, WriteVar:=STRUCT_UNION_ARR_D2_E1);
			264: iFileWriteVar(Execute:=TRUE, WriteVar:=STRUCT_UNION_ARR_D3_E1);

			// Alignment1Union
			300: iFileWriteVar(Execute:=TRUE, WriteVar:=UNION_ALIGNMENT1.Bytes);
			301: iFileWriteVar(Execute:=TRUE, WriteVar:=UNION_ALIGNMENT1_ARR_D1);
			
			// Alignment2Union
			310: iFileWriteVar(Execute:=TRUE, WriteVar:=UNION_ALIGNMENT2.Words);
			311: iFileWriteVar(Execute:=TRUE, WriteVar:=UNION_ALIGNMENT2_ARR_D1);
			312: iFileWriteVar(Execute:=TRUE, WriteVar:=UNION_ALIGNMENT2_ARR_D2);
			313: iFileWriteVar(Execute:=TRUE, WriteVar:=UNION_ALIGNMENT2_ARR_D3);
			314: iFileWriteVar(Execute:=TRUE, WriteVar:=UNION_ALIGNMENT2_ARR_D1_E1);
			315: iFileWriteVar(Execute:=TRUE, WriteVar:=UNION_ALIGNMENT2_ARR_D2_E1);
			316: iFileWriteVar(Execute:=TRUE, WriteVar:=UNION_ALIGNMENT2_ARR_D3_E1);
			
			// Alignment4Union
			320: iFileWriteVar(Execute:=TRUE, WriteVar:=UNION_ALIGNMENT4.Dwords);
			321: iFileWriteVar(Execute:=TRUE, WriteVar:=UNION_ALIGNMENT4_ARR_D1_E1);
			322: iFileWriteVar(Execute:=TRUE, WriteVar:=UNION_ALIGNMENT4_ARR_D2_E1);
			323: iFileWriteVar(Execute:=TRUE, WriteVar:=UNION_ALIGNMENT4_ARR_D3_E1);

			// Alignment8Union
			330: iFileWriteVar(Execute:=TRUE, WriteVar:=UNION_ALIGNMENT8.aLword);
			331: iFileWriteVar(Execute:=TRUE, WriteVar:=UNION_ALIGNMENT8_ARR_D1_E1);
			332: iFileWriteVar(Execute:=TRUE, WriteVar:=UNION_ALIGNMENT8_ARR_D2_E1);
			333: iFileWriteVar(Execute:=TRUE, WriteVar:=UNION_ALIGNMENT8_ARR_D3_E1);

			// ComplexStruct
			340: iFileWriteVar(Execute:=TRUE, WriteVar:=STRUCT_COMPLEX);

			// Nest3Struct
			350: iFileWriteVar(Execute:=TRUE, WriteVar:=STRUCT_NEST3);

			// ExampleStruct
			360: iFileWriteVar(Execute:=TRUE, WriteVar:=STRUCT_EXAMPLE);

			// ExampleUnion
			370: iFileWriteVar(Execute:=TRUE, WriteVar:=UNION_EXAMPLE.StatusCode);
		ELSE
			Inc(iState);
		END_CASE;
		
		IF iFileWriteVar.Done THEN
			Inc(iState);
		END_IF;
	27:
		iFileWriteVar(Execute:=FALSE, WriteVar:=iVarBin);
		
		Clear(iVarName);
		Clear(iVarDeclare);
		Clear(iVarValue);
		Clear(iVarKsType);
		Clear(iVarKsId);
		
		iState := iState - 5;
	29:
		iState := STATE_FINALIZE;

	// STATE_FINALIZE
	900:
		iFileWriter.Enable := FALSE;
		
		Inc(iState);
	901:
		IF NOT iFileWriter.Busy THEN
			iState := iState + 8;
		END_IF;
	909:
		iState := STATE_DONE;
	
	// STATE_DONE
	1000:
		Inc(iState);
END_CASE;

iFileWriter(Context:=iFileWriterContext,
			BufferContext:=iBufferContext,
			Buffer:=iBuffer);
END_PROGRAM

FUNCTION RingBuffer_writeAsHexStr : BOOL
VAR
    HEX_DIGITS : ARRAY[0..15] OF BYTE := [16#30, 16#31, 16#32, 16#33, 16#34, 16#35, 16#36, 16#37, 16#38, 16#39, 16#41, 16#42, 16#43, 16#44, 16#45, 16#46];
    iTerm : UINT;
    iTmp : ARRAY[0..1023] OF BYTE;
    iTmpHead : UINT;
    iChunk : ARRAY[0..15] OF BYTE;
    iChunkSize : UINT;
    iCharUpperIndex : UINT;
    iCharLowerIndex : UINT;
    iFlushInterval : UINT;
    iJoinSize : UINT;
    iChar : BYTE;
    i : UINT;
    j : UINT;
END_VAR
VAR_IN_OUT
    Context : stfreakjp\buf\RingBufferContext;
    Buffer : ARRAY[*] OF BYTE;
    In : ARRAY[*] OF BYTE;
END_VAR
VAR_INPUT
    Head : UINT := 0;
    Size : UINT := 0;
    Prefix : STRING[4] := '0x';
    Join : STRING[4] := ',';
    AllowOverwrite : BOOL := False;
END_VAR
VAR_OUTPUT
    WriteSize : UINT;
END_VAR
RingBuffer_writeAsHexStr := FALSE;
WriteSize := 0;
IF NOT EN THEN	
	RETURN;
END_IF;

iChunkSize := StringToAry(In:=Prefix, AryOut:=iChunk[0]);
iCharUpperIndex := iChunkSize;
iCharLowerIndex := iChunkSize + 1;
iJoinSize := StringToAry(In:=Join, AryOut:=iChunk[iChunkSize + 2]);
iChunkSize := iChunkSize + 2 + iJoinSize;

iFlushInterval := SizeOfAry(iTmp) / iChunkSize;
iTmpHead := 0;

iTerm := Head + Size;
i := Head;
j := iFlushInterval;
WHILE i < iTerm DO
	iChar := In[i];
	iChunk[iCharUpperIndex] := HEX_DIGITS[TO_UINT(SHR(iChar, 4) AND BYTE#16#0F)];
	iChunk[iCharLowerIndex] := HEX_DIGITS[TO_UINT(iChar AND BYTE#16#0F)];
	MemCopy(In:=iChunk[0], AryOut:=iTmp[iTmpHead], Size:=iChunkSize);
	iTmpHead := iTmpHead + iChunkSize;
	
	Inc(i);
	Dec(j);
	
	IF j < 1 THEN
		IF iTerm - i < 1 THEN
			iTmpHead := iTmpHead - iJoinSize;
		END_IF;
		IF NOT \\stfreakjp\buf\RingBuffer_write(Context:=Context,
												Buffer:=Buffer,
												In:=iTmp,
												Head:=0,
												Size:=iTmpHead,
												AllowOverwrite:=AllowOverwrite)
		THEN
			WriteSize := iChunkSize * (i - Head - 1);
			
			RETURN;
		END_IF;
		iTmpHead := 0;
		j := iFlushInterval;
	END_IF;
END_WHILE;
IF iTmpHead > 0 THEN
	iTmpHead := iTmpHead - iJoinSize;
	RingBuffer_writeAsHexStr :=
		\\stfreakjp\buf\RingBuffer_write(Context:=Context,
										 Buffer:=Buffer,
										 In:=iTmp,
										 Head:=0,
										 Size:=iTmpHead,
										 AllowOverwrite:=AllowOverwrite);
ELSE
	RingBuffer_writeAsHexStr := TRUE;
END_IF;

IF RingBuffer_writeAsHexStr THEN
	WriteSize := iChunkSize * Size - iJoinSize;
END_IF;
END_FUNCTION

FUNCTION RingBuffer_writeStr : BOOL
VAR
    iBin : ARRAY[0..4095] OF BYTE;
    iSize : UINT;
END_VAR
VAR_IN_OUT
    Context : stfreakjp\buf\RingBufferContext;
    Buffer : ARRAY[*] OF BYTE;
END_VAR
VAR_INPUT
    In : STRING[1986] := '';
    AllowOverwrite : BOOL := False;
END_VAR
VAR_OUTPUT
    WriteSize : UINT;
END_VAR
RingBuffer_writeStr := FALSE;
WriteSize := 0;
IF NOT EN THEN
	RETURN;
END_IF;

iSize := StringToAry(In:=In, AryOut:=iBin[0]);

IF \\stfreakjp\buf\RingBuffer_write(Context:=Context,
									Buffer:=Buffer,
									In:=iBin,
									Head:=0,
									Size:=iSize,
									AllowOverwrite:=AllowOverwrite)
THEN
	WriteSize := iSize;
	RingBuffer_writeStr := TRUE;
END_IF;
END_FUNCTION